(* Logix 5000 project; controller project2 vendor 1 type 14 code 54 rev 20.19; software revision 20.05 *)

TASK MainTask (continuous, watchdog 500 ms) : MainProgram

MODULES
   Local : vendor 1 type 14 code 54 (ICP 0, rev 20.19)
      fifth_module : 1756-OB32 (ICP 5, rev 3.2, Output RPI 20 ms)
      ENBT : 1756-ENBT (ICP 1, Ethernet 192.168.1.2, rev 4.3)
END_MODULES

VAR_GLOBAL   (* controller tags *)
   TAG_1_CONT : DINT := 16640;
END_VAR

PROGRAM MainProgram   (* main routine MainRoutine *)
VAR
   TAG_1_P_MAIN : DINT;
   TAG_2_P_MAIN : DINT := 2048;
   TAG_3_P_MAIN : DINT := 1;
   TAG_4_MP : INT;
END_VAR

ROUTINE MainRoutine   (* ladder *)
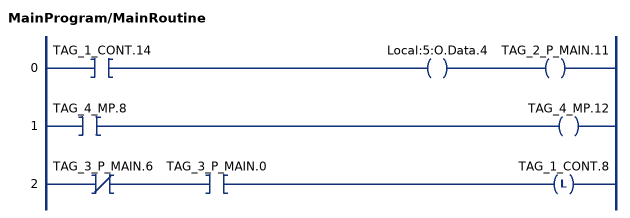
   0: XIC(TAG_1_CONT.14)OTE(Local:5:O.Data.4)OTE(TAG_2_P_MAIN.11);
   1: XIC(TAG_4_MP.8)OTE(TAG_4_MP.12);
   2: XIO(TAG_3_P_MAIN.6)XIC(TAG_3_P_MAIN.0)OTL(TAG_1_CONT.8);
END_ROUTINE
END_PROGRAM

PROGRAM PROG_2   (* main routine Routine1_PROG2 *)
VAR
   TAG_1_PROG2 : DINT := 1179010630;
   TAG_2_PROG2 : DINT;
END_VAR

ROUTINE Routine1_PROG2   (* ladder *)
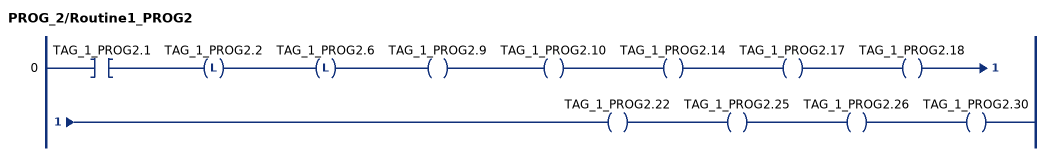
   0: XIC(TAG_1_PROG2.1)OTL(TAG_1_PROG2.2)OTL(TAG_1_PROG2.6)OTE(TAG_1_PROG2.9)OTE(TAG_1_PROG2.10)OTE(TAG_1_PROG2.14)OTE(TAG_1_PROG2.17)OTE(TAG_1_PROG2.18)OTE(TAG_1_PROG2.22)OTE(TAG_1_PROG2.25)OTE(TAG_1_PROG2.26)OTE(TAG_1_PROG2.30);
END_ROUTINE
END_PROGRAM
